// SIMATIC S7-200 project (STEP 7-Micro/WIN), CPU 222 CN REL 02.01

SYMBOL_TABLE 用户定义1
start            I1.0
END_SYMBOL_TABLE

ORGANIZATION_BLOCK 主程序:OB1
TITLE=PLC在首次上电时，调用PID定义子程序，设置PID的各项参数、配置高速计数器、初始化高速计数器、设置定时器间隔并附加PID执行中断。
// 当操作员按下启动按钮，系统启动电机并启用中断控制。
// 随后，PID执行中断定期触发，PLC读取高速计数器当前值，计算过程变量，与设定值比较，通过PID算法调整输出，最终更新变频器控制输出调节频率。
// 当停止按钮按下时，系统停止电机和中断控制。
// 当电机运行状态关闭时，系统断开中断并清零变频器控制输出，防止变频器继续运行。
// 为主程序保持转速控制的准确性，系统监控当前转速是否变化，若变化则更新设定值和上次转速。
// 电机运行启动时，附加PID执行中断，启用中断控制。
// 
BEGIN
Network 1 // 网络标题
// 网络注释
LD     SM0.1
CALL   PID定义:SBR0
Network 2
LD     start:I1.0
S      Q1.0, 1
S      Q1.2, 1
Network 3
LD     I1.1
R      Q1.0, 3
Network 4
LDR<>  VD0, VD4
MOVR   VD0, VD104
/R     50.0, VD104
MOVR   VD0, VD4
Network 5
LD     Q1.0
ED
DTCH   10
MOVW   0, AQW0
Network 6
LD     Q1.0
EU
ATCH   INT_0:INT0, 10
END_ORGANIZATION_BLOCK

SUBROUTINE_BLOCK PID定义:SBR0
TITLE=子程序注释
BEGIN
Network 1 // 网络标题
// 网络注释
LD     SM0.0
MOVR   0.5, VD104
MOVR   0.5, VD112
MOVR   0.1, VD116
MOVR   0.02, VD120
MOVR   0.0, VD124
Network 2
LD     SM0.0
MOVB   16#F8, SMB37
MOVD   0, SMD38
MOVD   0, SMD42
HDEF   0, 0
HSC    0
MOVB   250, SMB34
ATCH   INT_0:INT0, 10
ENI
END_SUBROUTINE_BLOCK

INTERRUPT_BLOCK INT_0:INT0
TITLE=中断程序注释
BEGIN
Network 1 // 网络标题
// 网络注释
LD     SM0.0
DTR    HC0, AC1
HSC    0
*R     240.0, AC1
MOVR   AC1, VD20
/R     500.0, VD20
MOVR   VD20, VD100
/R     1495.0, VD100
Network 2
LD     SM0.0
PID    VB100, 0
Network 3
LD     SM0.0
MOVR   VD108, AC0
*R     32000.0, AC0
ROUND  AC0, AC0
DTI    AC0, AQW0
END_INTERRUPT_BLOCK
